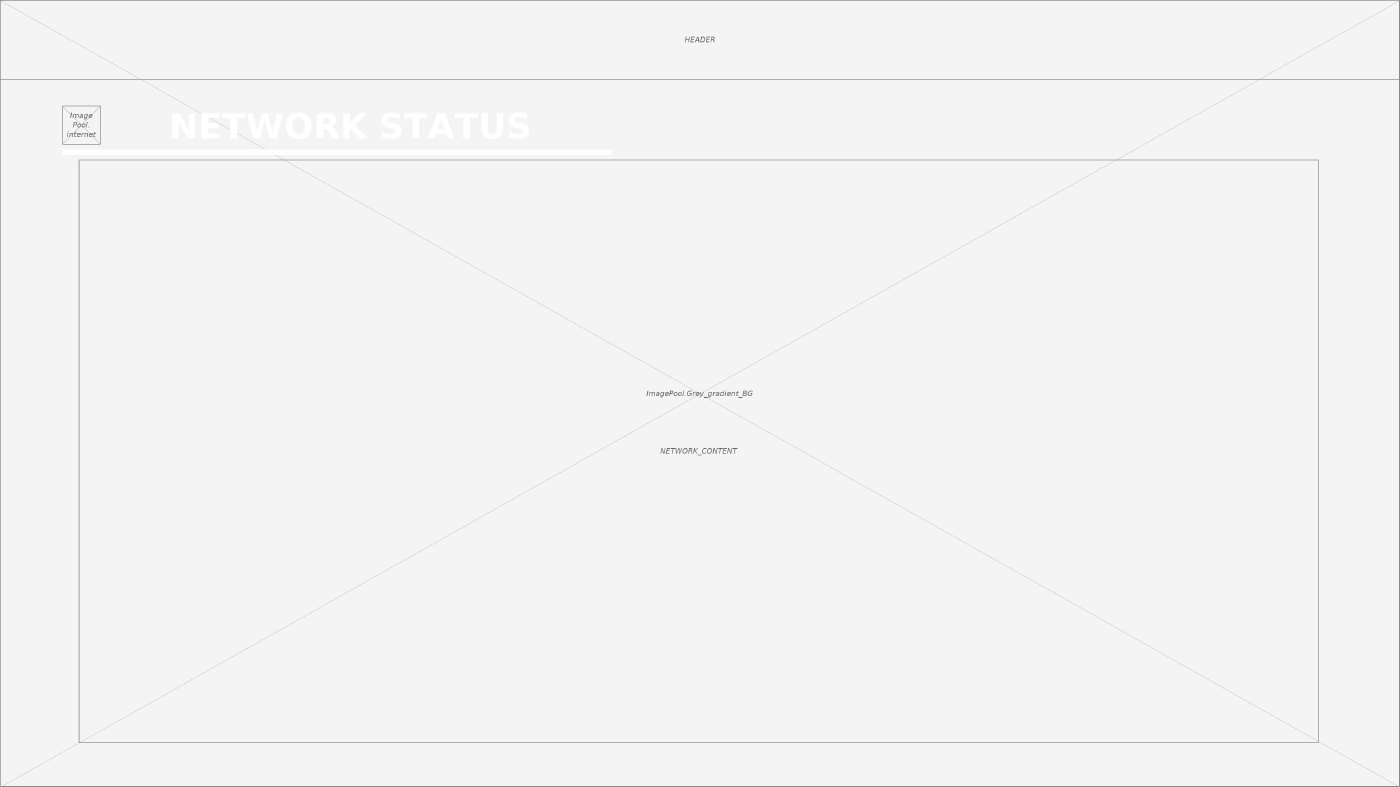
VISUALIZATION NETWORK_PAGE  // 1920x1080
    Image (0,0 1920x1080), image: ImagePool.Grey_gradient_BG
    Frame (0,0 1920x109)
        shows HEADER()
    Rectangle (143,136 675x74), "NETWORK STATUS"
    Rectangle (86,205 752x7)
    Image (85,145 53x53), image: ImagePool.internet
    Frame (108,219 1700x800)
        shows NETWORK_CONTENT()
END_VISUALIZATION

(* stored: Version 1.1.0.1, ProductVersion 3.1.4024.12
   Visu NETWORK_PAGE: Id {66f7206a-bce2-43f2-8daa-3d57922d930d} *)
